// The composition root: what is registered, what reports it, and the run that
// drives it.
//
// This is also a WORKED EXAMPLE. It composes the library the way a real project
// should - a run, a suite, three sinks - so anything awkward here is awkward for
// everyone.
//
// READ THESE, in the online view:
//
//   Complete   TRUE once every test has finished
//   Outcome    Passed if the library is sound
//   Total      111 - assert this. A test that stops being registered vanishes
//              silently, and CI sees fewer passes rather than a failure
//   Passed / Failed / Errors / Skipped
//   Idle       TRUE once the result document has reached disk. CI MUST WAIT FOR
//              BOTH Complete AND Idle - a run finishing and its file landing are
//              different events, and copying between them yields a truncated
//              artifact that reads as a broken pipeline
//
// WHERE A FAILURE SHOWS UP:
//   - the Logged Events window, as a log line and as an event
//   - C:\ProgramData\Beckhoff\TwinCAT\3.1\Boot\TestHarnessCoreResults.xml
//
// Read the failure there rather than from journal internals in a watch window.
// Making that unnecessary is what this library is for.
//
// THE FAILURE PATH IS EXERCISED, not assumed. The Verdict tests drive DELIBERATE
// failures into a private journal; the Suite tests register doubles that fail and
// error on purpose; the JUnit tests write to a folder that does not exist. They all
// pass. What they prove is that going wrong works.
//
// THE CHARACTERIZATION TESTS ARE THE ACCEPTANCE CONTRACT - behaviour a project
// depending on this library is entitled to rely on. They are also the only tests
// that ask questions of the ARTIFACT: how many cases the document carries, what
// type attribute a failure got, whether a timeout message names the wall clock.
//
// MULTI-SCAN TESTS hold a private runner, suite or run and step it one scan per
// call, returning FALSE until it finishes - the same mechanism they are verifying,
// one level down. Each carries a watchdog, so a defect that never completes fails
// its own test rather than hanging everything and looking like a broken verifier.
PROGRAM PRG_UnitTests
VAR
	// A RUN, not just a suite. RunFinished is a run-level event and only a TestRun
	// raises it - which is what produces a document at all.
	Runner : TestRun<2>;
	Suite  : TestSuite<130>;

	// All three sinks, which is the realistic composition: a log line to read at a
	// glance, an event to filter and route, a document for CI.
	LogSink	  : TestLogReporter;
	EventSink : TestEventReporter;
	JUnitSink : TestJUnitReporter;

	// The 4026 boot folder. Named apart from the files the JUnit tests write, so a
	// stale artifact from either cannot be mistaken for the other.
	ResultPath : T_MaxString := 'C:\ProgramData\Beckhoff\TwinCAT\3.1\Boot\TestHarnessCoreResults.xml';

	Budgets : ST_TestBudgets;
	Wired	: BOOL;

	// -- Registry --
	registryCapacityAndOverflow	: TEST_RegistryCapacityAndOverflow;
	registryRejectsDuplicateLabel	: TEST_RegistryRejectsDuplicateLabel;
	registryRejectsEmptyLabelAndNullTest	: TEST_RegistryRejectsEmptyLabelAndNullTest;
	registryClosesRegistration	: TEST_RegistryClosesRegistration;
	registryLookup	: TEST_RegistryLookup;
	registryPreservesOrder	: TEST_RegistryPreservesOrder;
	registrySlotCarriesItsIndex	: TEST_RegistrySlotCarriesItsIndex;
	registryResolvesOptionalHooks	: TEST_RegistryResolvesOptionalHooks;
	registryJournalsArePerSlot	: TEST_RegistryJournalsArePerSlot;
	registryJournalRejectsBadIndex	: TEST_RegistryJournalRejectsBadIndex;

	// -- Arbiter --
	arbiterVisitsEveryTestOnce	: TEST_ArbiterVisitsEveryTestOnce;
	arbiterCurrentIsNullWhenNothingActive	: TEST_ArbiterCurrentIsNullWhenNothingActive;
	arbiterEmptyPassIsComplete	: TEST_ArbiterEmptyPassIsComplete;
	arbiterAbandonEndsThePass	: TEST_ArbiterAbandonEndsThePass;
	arbiterNotExhaustedWhileLastTestRuns	: TEST_ArbiterNotExhaustedWhileLastTestRuns;
	arbiterRestartsFromTheBeginning	: TEST_ArbiterRestartsFromTheBeginning;

	// -- Verdict --
	verdictRecordsAFailure	: TEST_VerdictRecordsAFailure;
	verdictPassDoesNotOvertakeAFailure	: TEST_VerdictPassDoesNotOvertakeAFailure;
	verdictZeroChecksIsErrored	: TEST_VerdictZeroChecksIsErrored;
	verdictReportErrorIsNotAFailure	: TEST_VerdictReportErrorIsNotAFailure;
	verdictFailIsAPlainFailure	: TEST_VerdictFailIsAPlainFailure;
	verdictSummaryLeadsWithTheStepLabel	: TEST_VerdictSummaryLeadsWithTheStepLabel;
	verdictFirstFailureWinsTheSummary	: TEST_VerdictFirstFailureWinsTheSummary;
	verdictUntargetedHandleIsInert	: TEST_VerdictUntargetedHandleIsInert;

	// -- Journal --
	journalTimesOutOnCycles	: TEST_JournalTimesOutOnCycles;
	journalZeroBudgetDisablesTheDeadline	: TEST_JournalZeroBudgetDisablesTheDeadline;
	journalDefaultsFillOnlyWhatWasNotClaimed	: TEST_JournalDefaultsFillOnlyWhatWasNotClaimed;
	journalResetKeepsWhatWasRegistered	: TEST_JournalResetKeepsWhatWasRegistered;
	journalSkippedIsTerminalAndNotRed	: TEST_JournalSkippedIsTerminalAndNotRed;

	// -- Runner --
	runnerDrivesThePhasesInOrder	: TEST_RunnerDrivesThePhasesInOrder;
	runnerRunsAMultiScanBody	: TEST_RunnerRunsAMultiScanBody;
	runnerSetupFailureSkipsTheBody	: TEST_RunnerSetupFailureSkipsTheBody;
	runnerSetupDoesNotSpendTheBodyBudget	: TEST_RunnerSetupDoesNotSpendTheBodyBudget;
	runnerBodyDeadlineFires	: TEST_RunnerBodyDeadlineFires;
	runnerSetupDeadlineFires	: TEST_RunnerSetupDeadlineFires;
	runnerTeardownOverrunKeepsTheVerdict	: TEST_RunnerTeardownOverrunKeepsTheVerdict;
	runnerAbandonMakesOneFinalCall	: TEST_RunnerAbandonMakesOneFinalCall;
	runnerRefusesAnEmptySlot	: TEST_RunnerRefusesAnEmptySlot;

	// -- Suite --
	suiteRunsEveryRegisteredTest	: TEST_SuiteRunsEveryRegisteredTest;
	suiteSeparatesFailuresFromErrors	: TEST_SuiteSeparatesFailuresFromErrors;
	suiteClosesRegistrationOnFirstEnable	: TEST_SuiteClosesRegistrationOnFirstEnable;
	suiteRejectedRegistrationIsNeverSilent	: TEST_SuiteRejectedRegistrationIsNeverSilent;
	suiteSkipMarksEverythingSkipped	: TEST_SuiteSkipMarksEverythingSkipped;
	suiteSkippedAfterARejectedRegistrationIsErrored	: TEST_SuiteSkippedAfterARejectedRegistrationIsErrored;
	suiteSkippedWithNoLabelIsAFrameworkError	: TEST_SuiteSkippedWithNoLabelIsAFrameworkError;
	suiteReRunRepeatsTheRegisteredSet	: TEST_SuiteReRunRepeatsTheRegisteredSet;
	suiteReRunSingleRecordsNothing	: TEST_SuiteReRunSingleRecordsNothing;
	suiteWithNothingRegisteredIsComplete	: TEST_SuiteWithNothingRegisteredIsComplete;
	suiteWithNoLabelIsAFrameworkError	: TEST_SuiteWithNoLabelIsAFrameworkError;
	suiteDefaultsReachTheTests	: TEST_SuiteDefaultsReachTheTests;

	runAnnouncesItselfBeforeAnythingElse	: TEST_RunAnnouncesItselfBeforeAnythingElse;
	runRefusingASuiteIsNeverSilent	: TEST_RunRefusingASuiteIsNeverSilent;
	runPassesWithSkipsBesideAPass	: TEST_RunPassesWithSkipsBesideAPass;
	runOfOnlySkippedTestsIsSkipped	: TEST_RunOfOnlySkippedTestsIsSkipped;
	runWithMoreSkipsThanPassesIsPassed	: TEST_RunWithMoreSkipsThanPassesIsPassed;
	runReportsASuiteSkippedBeforeItsReporters	: TEST_RunReportsASuiteSkippedBeforeItsReporters;
	runReportsASkippedSuiteInItsPlace	: TEST_RunReportsASkippedSuiteInItsPlace;
	runReportsEachSkippedTestByName	: TEST_RunReportsEachSkippedTestByName;
	runReRunDoesNotRunASkippedSuite	: TEST_RunReRunDoesNotRunASkippedSuite;
	runReRunReportsASkippedSuiteAgain	: TEST_RunReRunReportsASkippedSuiteAgain;

	// -- Fanout --
	fanoutNotifiesEverySinkInOrder	: TEST_FanoutNotifiesEverySinkInOrder;
	fanoutOnlyChecksGoToDetailSinks	: TEST_FanoutOnlyChecksGoToDetailSinks;
	fanoutIsIdleIsTheAndOfEverySink	: TEST_FanoutIsIdleIsTheAndOfEverySink;
	fanoutSuspendSilencesEverything	: TEST_FanoutSuspendSilencesEverything;
	fanoutRefusesBeyondCapacityAndTellsTheRest	: TEST_FanoutRefusesBeyondCapacityAndTellsTheRest;
	fanoutCarriesTheSuiteResultThrough	: TEST_FanoutCarriesTheSuiteResultThrough;

	fanoutForwardsRunStarted	: TEST_FanoutForwardsRunStarted;

	// -- LogReporter --
	logReporterIsQuietAboutPasses	: TEST_LogReporterIsQuietAboutPasses;
	logReporterWritesFailuresAndErrors	: TEST_LogReporterWritesFailuresAndErrors;
	logReporterNarratesWhenAsked	: TEST_LogReporterNarratesWhenAsked;
	logReporterAlwaysWritesFrameworkErrors	: TEST_LogReporterAlwaysWritesFrameworkErrors;
	logReporterSummarisesASuite	: TEST_LogReporterSummarisesASuite;
	logReporterNarratesSkipsOnlyWhenAsked	: TEST_LogReporterNarratesSkipsOnlyWhenAsked;
	logReporterNamesASkippedAndAnErroredRun	: TEST_LogReporterNamesASkippedAndAnErroredRun;

	jUnitReporterOpensOnRunStarted	: TEST_JUnitReporterOpensOnRunStarted;

	// -- EventReporter --
	eventReporterSendsAndDoesNotFail	: TEST_EventReporterSendsAndDoesNotFail;
	eventReporterIsQuietAboutPasses	: TEST_EventReporterIsQuietAboutPasses;
	eventReporterRaisesEachOutcomeOnce	: TEST_EventReporterRaisesEachOutcomeOnce;
	eventReporterWorksThroughTheFanout	: TEST_EventReporterWorksThroughTheFanout;
	eventReporterDoesNotCallASkipAPass	: TEST_EventReporterDoesNotCallASkipAPass;
	eventReporterNamesASkippedAndAnErroredRun	: TEST_EventReporterNamesASkippedAndAnErroredRun;

	// -- JUnitReporter --
	jUnitReporterWritesTheDocument	: TEST_JUnitReporterWritesTheDocument;
	jUnitReporterIsBusyWhileWriting	: TEST_JUnitReporterIsBusyWhileWriting;
	jUnitReporterReportsAFailedWrite	: TEST_JUnitReporterReportsAFailedWrite;
	jUnitReporterRefusesWithNoPath	: TEST_JUnitReporterRefusesWithNoPath;
	jUnitReporterWritesNothingWhenNothingRan	: TEST_JUnitReporterWritesNothingWhenNothingRan;

	// -- Pure functions: the comparison and rendering rules --
	compareNumericRules	: TEST_CompareNumericRules;
	compareTextRules	: TEST_CompareTextRules;
	compareOtherRules	: TEST_CompareOtherRules;
	summaryLineComposition	: TEST_SummaryLineComposition;
	valueRendering	: TEST_ValueRendering;
	valueBriefShortens	: TEST_ValueBriefShortens;

	// -- Assertions: the public surface every user touches --
	assertNotEqualRejectsSameness	: TEST_AssertNotEqualRejectsSameness;
	assertGreaterAndLessCompareTheRightWayRound	: TEST_AssertGreaterAndLessCompareTheRightWayRound;
	assertNearUsesAbsoluteTolerance	: TEST_AssertNearUsesAbsoluteTolerance;
	assertWithinUsesRelativeTolerance	: TEST_AssertWithinUsesRelativeTolerance;
	assertInRangeIsInclusive	: TEST_AssertInRangeIsInclusive;
	assertBufferComparisons	: TEST_AssertBufferComparisons;
	assertCompletedWithinCountsCompletedScans	: TEST_AssertCompletedWithinCountsCompletedScans;

	stopwatchMeasuresAndFreezes	: TEST_StopwatchMeasuresAndFreezes;
	registeredAndReporterCountsAreReadable	: TEST_RegisteredAndReporterCountsAreReadable;
	// -- Suite watchdog --
	watchdogAbandonsAStalledSuite	: TEST_WatchdogAbandonsAStalledSuite;
	watchdogMeasuresProgressNotTime	: TEST_WatchdogMeasuresProgressNotTime;
	watchdogZeroDisablesIt	: TEST_WatchdogZeroDisablesIt;

	// -- Characterization: the acceptance contract --
	cHAR_Capacity	: CHAR_Capacity;
	cHAR_OverflowStatistics	: CHAR_OverflowStatistics;
	cHAR_ReRunTests	: CHAR_ReRunTests;
	cHAR_ReRunIndividual	: CHAR_ReRunIndividual;
	cHAR_WallClockTimeout	: CHAR_WallClockTimeout;
	cHAR_TimeoutPrecedence	: CHAR_TimeoutPrecedence;
	cHAR_SerialExecution	: CHAR_SerialExecution;

	// -- the result, for the watch window ---------------------------------------
	Complete : BOOL;
	Outcome	 : E_RunOutcome;
	Total	 : UDINT;
	Passed	 : UDINT;
	Failed	 : UDINT;
	Errors	 : UDINT;
	Skipped	 : UDINT;
	Duration : LREAL;

	// -- did the artifact land? -------------------------------------------------
	Idle		  : BOOL;
	FilesWritten  : UDINT;
	WriteFailures : UDINT;
END_VAR

IF NOT Wired THEN
	Wired := TRUE;

	Suite.SetLabel('TestHarnessCore');

	// Registry
	Suite.Register(registryCapacityAndOverflow, 'Registry: capacity and overflow', Budgets);
	Suite.Register(registryRejectsDuplicateLabel, 'Registry: rejects a duplicate label', Budgets);
	Suite.Register(registryRejectsEmptyLabelAndNullTest, 'Registry: rejects an empty label and a null test', Budgets);
	Suite.Register(registryClosesRegistration, 'Registry: closes registration on first enable', Budgets);
	Suite.Register(registryLookup, 'Registry: lookup by label', Budgets);
	Suite.Register(registryPreservesOrder, 'Registry: preserves registration order', Budgets);
	Suite.Register(registrySlotCarriesItsIndex, 'Registry: a slot carries its own index', Budgets);
	Suite.Register(registryResolvesOptionalHooks, 'Registry: resolves the optional hooks independently', Budgets);
	Suite.Register(registryJournalsArePerSlot, 'Registry: journals are per slot and live', Budgets);
	Suite.Register(registryJournalRejectsBadIndex, 'Registry: an out-of-range journal is invalid', Budgets);

	// Arbiter
	Suite.Register(arbiterVisitsEveryTestOnce, 'Arbiter: visits every test once, in order', Budgets);
	Suite.Register(arbiterCurrentIsNullWhenNothingActive, 'Arbiter: current is null when nothing is active', Budgets);
	Suite.Register(arbiterEmptyPassIsComplete, 'Arbiter: an empty pass is complete, not stuck', Budgets);
	Suite.Register(arbiterAbandonEndsThePass, 'Arbiter: abandon does not visit the rest', Budgets);
	Suite.Register(arbiterNotExhaustedWhileLastTestRuns, 'Arbiter: not exhausted while the last test runs', Budgets);
	Suite.Register(arbiterRestartsFromTheBeginning, 'Arbiter: begin restarts from the first test', Budgets);

	// Verdict
	Suite.Register(verdictRecordsAFailure, 'Verdict: a mismatched check is recorded as a failure', Budgets);
	Suite.Register(verdictPassDoesNotOvertakeAFailure, 'Verdict: a pass cannot undo a failure', Budgets);
	Suite.Register(verdictZeroChecksIsErrored, 'Verdict: finishing with no checks is Errored', Budgets);
	Suite.Register(verdictReportErrorIsNotAFailure, 'Verdict: ReportError produces Errored, not Failed', Budgets);
	Suite.Register(verdictFailIsAPlainFailure, 'Verdict: Fail produces Failed', Budgets);
	Suite.Register(verdictSummaryLeadsWithTheStepLabel, 'Verdict: the summary leads with the step label', Budgets);
	Suite.Register(verdictFirstFailureWinsTheSummary, 'Verdict: the first failure wins the summary', Budgets);
	Suite.Register(verdictUntargetedHandleIsInert, 'Verdict: an untargeted handle records nothing', Budgets);

	// Journal
	Suite.Register(journalTimesOutOnCycles, 'Journal: a scan budget expires and records itself', Budgets);
	Suite.Register(journalZeroBudgetDisablesTheDeadline, 'Journal: a zero budget never expires', Budgets);
	Suite.Register(journalDefaultsFillOnlyWhatWasNotClaimed, 'Journal: defaults fill only unclaimed units', Budgets);
	Suite.Register(journalResetKeepsWhatWasRegistered, 'Journal: reset clears the verdict, keeps the budgets', Budgets);
	Suite.Register(journalSkippedIsTerminalAndNotRed, 'Journal: skipped is terminal and not a failure', Budgets);

	// Runner
	Suite.Register(runnerDrivesThePhasesInOrder, 'Runner: setup, body, teardown, each once, in order', Budgets);
	Suite.Register(runnerRunsAMultiScanBody, 'Runner: a multi-scan body is called until it finishes', Budgets);
	Suite.Register(runnerSetupFailureSkipsTheBody, 'Runner: a failed setup skips the body but not teardown', Budgets);
	Suite.Register(runnerSetupDoesNotSpendTheBodyBudget, 'Runner: setup does not spend the body scan budget', Budgets);
	Suite.Register(runnerBodyDeadlineFires, 'Runner: the body deadline stops a hanging test', Budgets);
	Suite.Register(runnerSetupDeadlineFires, 'Runner: setup has its own deadline', Budgets);
	Suite.Register(runnerTeardownOverrunKeepsTheVerdict, 'Runner: a teardown overrun does not change the verdict', Budgets);
	Suite.Register(runnerAbandonMakesOneFinalCall, 'Runner: abandon makes one final call and skips teardown', Budgets);
	Suite.Register(runnerRefusesAnEmptySlot, 'Runner: an empty slot is refused', Budgets);

	// Suite
	Suite.Register(suiteRunsEveryRegisteredTest, 'Suite: runs every registered test, once', Budgets);
	Suite.Register(suiteSeparatesFailuresFromErrors, 'Suite: failures and errors are counted apart', Budgets);
	Suite.Register(suiteClosesRegistrationOnFirstEnable, 'Suite: registration closes on first enable', Budgets);
	Suite.Register(suiteRejectedRegistrationIsNeverSilent, 'Suite: a rejected registration is never silent', Budgets);
	Suite.Register(suiteSkipMarksEverythingSkipped, 'Suite: Skip marks everything skipped and completes', Budgets);
	Suite.Register(suiteSkippedAfterARejectedRegistrationIsErrored, 'Suite: a registration refused before a skip is still counted', Budgets);
	Suite.Register(suiteSkippedWithNoLabelIsAFrameworkError, 'Suite: a skipped suite with no label is a framework error', Budgets);
	Suite.Register(suiteReRunRepeatsTheRegisteredSet, 'Suite: a re-run repeats the registered set', Budgets);
	Suite.Register(suiteReRunSingleRecordsNothing, 'Suite: an individual re-run records nothing', Budgets);
	Suite.Register(suiteWithNothingRegisteredIsComplete, 'Suite: an empty suite is complete, not red', Budgets);
	Suite.Register(suiteWithNoLabelIsAFrameworkError, 'Suite: an unnamed suite is a framework error', Budgets);
	Suite.Register(suiteDefaultsReachTheTests, 'Suite: suite defaults reach every unclaimed test', Budgets);

	Suite.Register(runAnnouncesItselfBeforeAnythingElse, 'Suite: a run announces itself before any result in it', Budgets);
	Suite.Register(runRefusingASuiteIsNeverSilent, 'Suite: a suite refused at composition still turns the run red', Budgets);
	Suite.Register(runPassesWithSkipsBesideAPass, 'Suite: a run with a pass and skips beside it is Passed', Budgets);
	Suite.Register(runOfOnlySkippedTestsIsSkipped, 'Suite: a run in which every test was skipped is Skipped', Budgets);
	Suite.Register(runWithMoreSkipsThanPassesIsPassed, 'Suite: a run with more skips than passes is still Passed', Budgets);
	Suite.Register(runReportsASuiteSkippedBeforeItsReporters, 'Suite: a suite skipped before its reporters were attached still reaches them', Budgets);
	Suite.Register(runReportsASkippedSuiteInItsPlace, 'Suite: a skipped suite is reported in its place in the run, not when Skip was called', Budgets);
	Suite.Register(runReportsEachSkippedTestByName, 'Suite: every skipped test reaches the sinks by name, before its suite closes', Budgets);
	Suite.Register(runReRunDoesNotRunASkippedSuite, 'Suite: a re-run does not run the tests of a skipped suite', Budgets);
	Suite.Register(runReRunReportsASkippedSuiteAgain, 'Suite: a re-run reports a skipped suite again, as skipped', Budgets);

	// Fanout
	Suite.Register(fanoutNotifiesEverySinkInOrder, 'Fanout: every sink is notified, in attachment order', Budgets);
	Suite.Register(fanoutOnlyChecksGoToDetailSinks, 'Fanout: only detail sinks receive checks', Budgets);
	Suite.Register(fanoutIsIdleIsTheAndOfEverySink, 'Fanout: IsIdle is the AND of every sink', Budgets);
	Suite.Register(fanoutSuspendSilencesEverything, 'Fanout: Suspend silences notifications but not CyclicLogic', Budgets);
	Suite.Register(fanoutRefusesBeyondCapacityAndTellsTheRest, 'Fanout: attachment beyond capacity is refused and reported', Budgets);
	Suite.Register(fanoutCarriesTheSuiteResultThrough, 'Fanout: SuiteFinished carries the live read model', Budgets);

	Suite.Register(fanoutForwardsRunStarted, 'Fanout: RunStarted reaches every sink and Suspend silences it', Budgets);

	// LogReporter
	Suite.Register(logReporterIsQuietAboutPasses, 'LogReporter: quiet about passes by default', Budgets);
	Suite.Register(logReporterWritesFailuresAndErrors, 'LogReporter: failures and errors are written and counted apart', Budgets);
	Suite.Register(logReporterNarratesWhenAsked, 'LogReporter: verbosity turns narration on and off', Budgets);
	Suite.Register(logReporterAlwaysWritesFrameworkErrors, 'LogReporter: framework errors are never suppressed', Budgets);
	Suite.Register(logReporterSummarisesASuite, 'LogReporter: one line per suite, carrying the counts', Budgets);
	Suite.Register(logReporterNarratesSkipsOnlyWhenAsked, 'LogReporter: a skip is narrated only when asked, and never as a failure', Budgets);
	Suite.Register(logReporterNamesASkippedAndAnErroredRun, 'LogReporter: a skipped run and an errored run each get their own banner', Budgets);

	Suite.Register(jUnitReporterOpensOnRunStarted, 'JUnitReporter: the document opens on RunStarted', Budgets);

	// EventReporter
	Suite.Register(eventReporterSendsAndDoesNotFail, 'EventReporter: an event is accepted and no HRESULT is returned', Budgets);
	Suite.Register(eventReporterIsQuietAboutPasses, 'EventReporter: quiet about passes until narration is asked for', Budgets);
	Suite.Register(eventReporterRaisesEachOutcomeOnce, 'EventReporter: one event per notification, none raised twice', Budgets);
	Suite.Register(eventReporterWorksThroughTheFanout, 'EventReporter: it sits behind the fan-out beside the log sink', Budgets);
	Suite.Register(eventReporterDoesNotCallASkipAPass, 'EventReporter: a skipped test raises no event, and never TestPassed', Budgets);
	Suite.Register(eventReporterNamesASkippedAndAnErroredRun, 'EventReporter: a skipped run and an errored run each raise their own event', Budgets);

	// JUnitReporter
	Suite.Register(jUnitReporterWritesTheDocument, 'JUnitReporter: the document reaches disk', Budgets);
	Suite.Register(jUnitReporterIsBusyWhileWriting, 'JUnitReporter: IsIdle is FALSE until the file lands', Budgets);
	Suite.Register(jUnitReporterReportsAFailedWrite, 'JUnitReporter: a failed write is counted and reported (R3)', Budgets);
	Suite.Register(jUnitReporterRefusesWithNoPath, 'JUnitReporter: no path set is a failure, not silence', Budgets);
	Suite.Register(jUnitReporterWritesNothingWhenNothingRan, 'JUnitReporter: an empty run produces no document', Budgets);

	// Pure functions - what equality and rendering MEAN. The object tests exercise
	// them incidentally, whenever some test happens to call AssertEqual, which is
	// not the same as pinning the rules themselves.
	Suite.Register(compareNumericRules, 'Pure: numeric rules: value across widths, exact floats, the hint', Budgets);
	Suite.Register(compareTextRules, 'Pure: string rules: content not capacity, and WSTRING as WSTRING (R1)', Budgets);
	Suite.Register(compareOtherRules, 'Pure: structs, arrays and enums; a size difference is a type difference', Budgets);
	Suite.Register(summaryLineComposition, 'Pure: composition order; the message is dropped whole, not cut', Budgets);
	Suite.Register(valueRendering, 'Pure: values render as something, including enums', Budgets);
	Suite.Register(valueBriefShortens, 'Pure: long values are shortened and marked', Budgets);

	// Assertions - the part of the library every user touches. Each of these checks
	// the direction that would be silently wrong, not just the happy path: a
	// reversed comparison passes every test written against it.
	Suite.Register(assertNotEqualRejectsSameness, 'Assertion: AssertNotEqual passes on difference, fails on sameness', Budgets);
	Suite.Register(assertGreaterAndLessCompareTheRightWayRound, 'Assertion: ordering runs the way the name says, both directions', Budgets);
	Suite.Register(assertNearUsesAbsoluteTolerance, 'Assertion: an absolute band, inclusive and symmetric', Budgets);
	Suite.Register(assertWithinUsesRelativeTolerance, 'Assertion: a relative band that holds across magnitudes', Budgets);
	Suite.Register(assertInRangeIsInclusive, 'Assertion: inclusive on both bounds', Budgets);
	Suite.Register(assertBufferComparisons, 'Assertion: byte offset, size mismatch, and a null buffer', Budgets);
	Suite.Register(assertCompletedWithinCountsCompletedScans, 'Assertion: the scan in progress is not counted', Budgets);

	Suite.Register(stopwatchMeasuresAndFreezes, 'Pure: the stopwatch advances, freezes and resets', Budgets);
	Suite.Register(registeredAndReporterCountsAreReadable, 'Suite: the counts CI is told to assert are readable', Budgets);
	// Suite watchdog - the run is the only object positioned to see a suite that
	// has stopped, because the suite IS the thing that stopped.
	Suite.Register(watchdogAbandonsAStalledSuite, 'Watchdog: a stalled suite is named, abandoned and counted', Budgets);
	Suite.Register(watchdogMeasuresProgressNotTime, 'Watchdog: a progressing suite is never abandoned, however slow', Budgets);
	Suite.Register(watchdogZeroDisablesIt, 'Watchdog: a zero budget never fires', Budgets);

	// Characterization - the acceptance contract. Behaviour a project depending on
	// this library is entitled to rely on, and the only tests that ask questions of
	// the result document rather than of a counter.
	Suite.Register(cHAR_Capacity, 'Contract: capacity holds what it says; overflow is reported', Budgets);
	Suite.Register(cHAR_OverflowStatistics, 'Contract: errors are counted apart from failures', Budgets);
	Suite.Register(cHAR_ReRunTests, 'Contract: one suite node per run; a re-run produces a fresh document', Budgets);
	Suite.Register(cHAR_ReRunIndividual, 'Contract: an individual re-run records nothing', Budgets);
	Suite.Register(cHAR_WallClockTimeout, 'Contract: the wall-clock deadline fires and names itself', Budgets);
	Suite.Register(cHAR_TimeoutPrecedence, 'Contract: suite default, per-test override, per-unit tracking', Budgets);
	Suite.Register(cHAR_SerialExecution, 'Contract: no test body runs while another is running', Budgets);

	// -- reporting -------------------------------------------------------------
	JUnitSink.SetPath(ResultPath);
	// Where a failed write is reported. Deliberately the log sink and not the
	// fan-out, which would call back into the writer that just failed.
	JUnitSink.AttachErrorSink(LogSink);

	Runner.SetLabel('TestHarnessCoreVerifier');
	// Which BUILD of the library ran, printed in both run banners and written to the
	// result document. The library is resolved as 'newest installed', so the build
	// under test is otherwise invisible. A version names an install, not its
	// contents: bump it for every build that needs telling apart, or two different
	// builds will print the same line.
	Runner.SetTargetInfo(CONCAT('TestHarnessCoreVerifier, library ',
								 TestHarnessCore.stLibVersion_TestHarnessCore.sVersion));

	// Attached to the RUN, which pushes each one into every suite. One attachment
	// point, whatever order suites and sinks are added in.
	Runner.AddReporter(LogSink);
	Runner.AddReporter(EventSink);
	Runner.AddReporter(JUnitSink);

	Runner.AddSuite(Suite);
END_IF

Runner.Run(Enable := TRUE);

// Read from the RUN, not the suite: it is the top of the nest, and the figures
// mean the same thing at every level.
Complete := Runner.IsComplete;
Outcome	 := Runner.Outcome;
Total	 := Runner.TestCount;
Passed	 := Runner.PassedCount;
Failed	 := Runner.FailedCount;
Errors	 := Runner.ErrorCount;
Skipped	 := Runner.SkippedCount;
Duration := Runner.TotalDuration;

Idle		  := JUnitSink.IsIdle;
FilesWritten  := JUnitSink.FilesWritten;
WriteFailures := JUnitSink.WriteFailures;

END_PROGRAM

(* stored: Version 1.1.0.1, ProductVersion 3.1.4026.18
   POU PRG_UnitTests: Id {09743738-8bdb-4d07-a6fb-ca1cd3adc3bb}, SpecialFunc None *)
